// TIA Portal project "Prog_Siemens_MPROT_V15.1" (V15.1)

(* hardware
DEVICE "S7-400 station_1"  S7-400 station
   slot 0: "UR1_0"  UR1  6ES7 400-1TA01-0AA0
   slot 1: "PS 407 4A_1"  PS 407 4A  6ES7 407-0DA02-0AA0
   slot 2: "S7-400"  CPU 414-3 PN/DP  6ES7 414-3EM05-0AB0  V5.1
      slot 2: "MPI/DP interface_1"  X1
      slot 5: "PROFINET interface_1"  PN-IO
         slot 1: "Port_1"  Port
         slot 2: "Port_2"  Port
   slot 4: "DO 16x24VDC/2A_1"  DO16 x 24VDC / 2A  6ES7 422-1BH11-0AA0
DEVICE "S7-1200 station_1"  S7-1200 Station
   slot 0: "Rack_0"  S7-1200 Rack  Rack  V1.0
   slot 1: "S7-1200"  CPU 1212C DC/DC/DC  6ES7 212-1AE31-0XB0  V3.0
*)

// ===== PLC "S7-400"  CPU 414-3 PN/DP =====

DATA_BLOCK "DB_Comunicacao"   // DB5
{ S7_Optimized_Access := 'FALSE' }
VERSION : 0.1
   VAR
      Valor_String : String[20] := 'Teste 400';
      Valor_Bit : Bool := True;
      Valor_Real : Real := 1234.567;
      Valor_Word : Word := 65535;
      Valor_Dword : DWord := 4294967295;
      Valor_Int : Int := -32767;
      Valor_Dint : DInt := -2147483647;
      Valor_Byte : Byte := 16#FF;
   END_VAR
BEGIN
END_DATA_BLOCK

ORGANIZATION_BLOCK "Main"   // OB1, LAD
TITLE = "Main Program Sweep (Cycle)"
{ S7_Optimized_Access := 'FALSE' }
VERSION : 0.1
   VAR_TEMP
      OB1_EV_CLASS : Byte;   // Bits 0-3 = 1 (Coming event), Bits 4-7 = 1 (Event class 1)
      OB1_SCAN_1 : Byte;   // 1 (Cold restart scan 1 of OB 1), 3 (Scan 2-n of OB 1)
      OB1_PRIORITY : Byte;   // Priority of OB Execution
      OB1_OB_NUMBR : Byte;   // 1 (Organization block 1, OB1)
      OB1_RESERVED_1 : Byte;   // Reserved for system
      OB1_RESERVED_2 : Byte;   // Reserved for system
      OB1_PREV_CYCLE : Int;   // Cycle time of previous OB1 scan (milliseconds)
      OB1_MIN_CYCLE : Int;   // Minimum cycle time of OB1 (milliseconds)
      OB1_MAX_CYCLE : Int;   // Maximum cycle time of OB1 (milliseconds)
      OB1_DATE_TIME : Date_And_Time;   // Date and time OB1 started
   END_VAR
BEGIN
END_ORGANIZATION_BLOCK

// ===== PLC "S7-1200"  CPU 1212C DC/DC/DC =====

DATA_BLOCK "DB_Comunicacao"   // DB3
{ S7_Optimized_Access := 'FALSE' }
VERSION : 0.1
   VAR
      Valor_String : String[20] := 'Teste 1200';
      Valor_Bit : Bool := True;
      Valor_Real : Real := 1234.567;
      Valor_Word : Word := 65535;
      Valor_Dword : DWord := 4294967295;
      Valor_Int : Int := -32767;
      Valor_DInt : DInt := -2147483647;
      Valor_Byte : Byte := 16#FF;
      Valor_DataHora : DTL := DTL#2020-06-21-08:51:32;
   END_VAR
BEGIN
END_DATA_BLOCK

ORGANIZATION_BLOCK "Main"   // OB1, LAD, ProgramCycle
TITLE = "Main Program Sweep (Cycle)"
{ S7_Optimized_Access := 'TRUE' }
VERSION : 0.1
BEGIN
END_ORGANIZATION_BLOCK